{attribute 'qualified_only'}
{attribute 'strict'}
TYPE EnumState :
(
	init,
	drive1,
	drive2,
	reset
);
END_TYPE

(* stored: Version 1.1.0.1, ProductVersion 3.1.4022.3
   DUT EnumState: Id {be140ba5-bd42-4dbc-880c-11c28c9d38f4} *)
